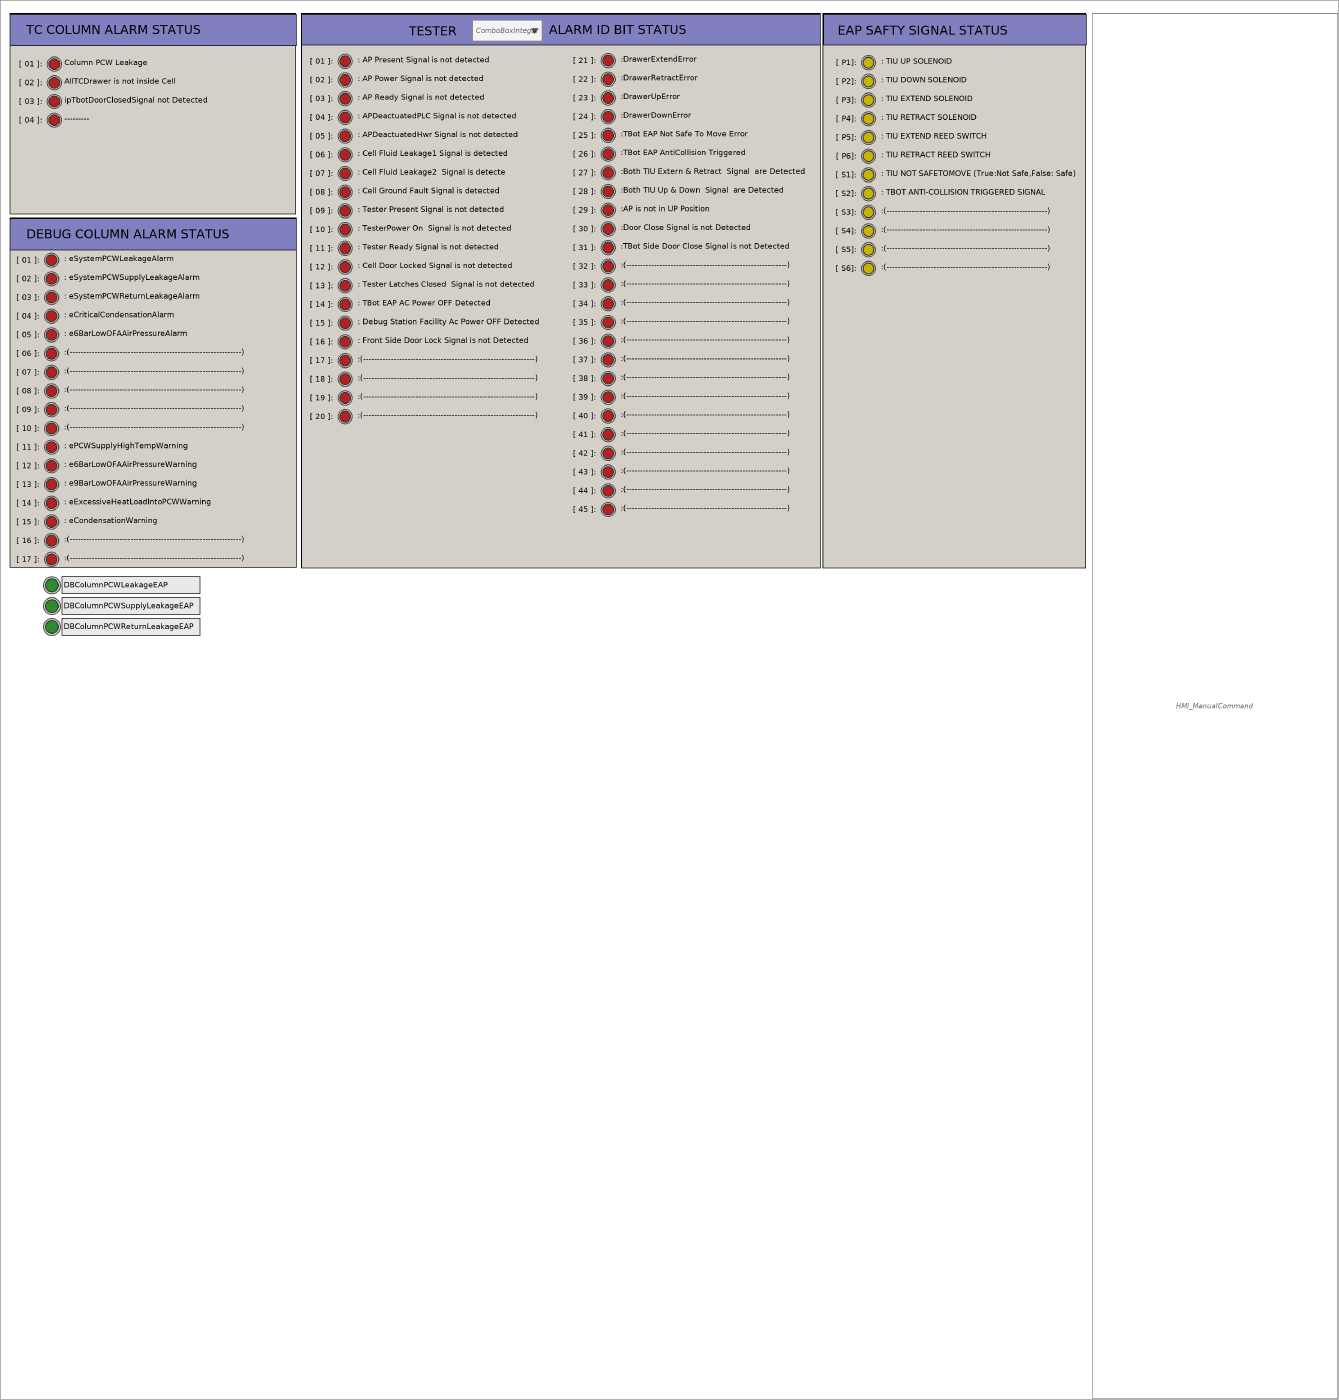
VISUALIZATION HMI_Alarm  // 1934x2021
    Rectangle (1188,19 380x801)
    Rectangle (1189,20 380x45)
    Rectangle (435,19 750x801)
    Rectangle (435,20 750x45)
    Rectangle (14,19 413x290)
    Rectangle (14,20 414x46)
    Lamp1 (866,75 25x25), variable: ALMTC.Level[iHMICbLevelSelection].AlarmID[21], style: Lamp-Lamp1-Red
    Label (824,75 40x25), "[ 21 ]:"
    Label (890,73 300x25), ":DrawerExtendError"
    ComboBoxInteger (682,29 101x30), variable: iHMICbLevelSelection, text list: 'LevelTxtList'
    Lamp1 (866,102 25x25), variable: ALMTC.Level[iHMICbLevelSelection].AlarmID[22], style: Lamp-Lamp1-Red
    Label (824,102 40x25), "[ 22 ]:"
    Label (890,100 300x25), ":DrawerRetractError"
    Lamp1 (866,129 25x25), variable: ALMTC.Level[iHMICbLevelSelection].AlarmID[23], style: Lamp-Lamp1-Red
    Label (824,129 40x25), "[ 23 ]:"
    Label (890,127 300x25), ":DrawerUpError"
    Lamp1 (866,156 25x25), variable: ALMTC.Level[iHMICbLevelSelection].AlarmID[24], style: Lamp-Lamp1-Red
    Label (824,156 40x25), "[ 24 ]:"
    Label (890,154 300x25), ":DrawerDownError"
    Lamp1 (866,183 25x25), variable: ALMTC.Level[iHMICbLevelSelection].AlarmID[25], style: Lamp-Lamp1-Red
    Label (824,183 40x25), "[ 25 ]:"
    Label (890,181 300x25), ":TBot EAP Not Safe To Move Error"
    Lamp1 (866,210 25x25), variable: ALMTC.Level[iHMICbLevelSelection].AlarmID[26], style: Lamp-Lamp1-Red
    Label (824,210 40x25), "[ 26 ]:"
    Label (890,208 300x25), ":TBot EAP AntiCollision Triggered"
    Lamp1 (866,237 25x25), variable: ALMTC.Level[iHMICbLevelSelection].AlarmID[27], style: Lamp-Lamp1-Red
    Label (824,237 40x25), "[ 27 ]:"
    Label (890,235 300x25), ":Both TIU Extern & Retract Signal are Detected"
    Lamp1 (866,264 25x25), variable: ALMTC.Level[iHMICbLevelSelection].AlarmID[28], style: Lamp-Lamp1-Red
    Label (824,264 40x25), "[ 28 ]:"
    Label (890,262 300x25), ":Both TIU Up & Down Signal are Detected"
    Lamp1 (866,291 25x25), variable: ALMTC.Level[iHMICbLevelSelection].AlarmID[29], style: Lamp-Lamp1-Red
    Label (824,291 40x25), "[ 29 ]:"
    Label (890,289 300x25), ":AP is not in UP Position"
    Lamp1 (866,318 25x25), variable: ALMTC.Level[iHMICbLevelSelection].AlarmID[30], style: Lamp-Lamp1-Red
    Label (824,318 40x25), "[ 30 ]:"
    Label (890,316 300x25), ":Door Close Signal is not Detected"
    Lamp1 (866,345 25x25), variable: ALMTC.Level[iHMICbLevelSelection].AlarmID[31], style: Lamp-Lamp1-Red
    Label (824,345 40x25), "[ 31 ]:"
    Label (890,343 300x25), ":TBot Side Door Close Signal is not Detected"
    Lamp1 (866,372 25x25), variable: ALMTC.Level[iHMICbLevelSelection].AlarmID[32], style: Lamp-Lamp1-Red
    Label (824,372 40x25), "[ 32 ]:"
    Label (890,370 300x25), ":(----------------------------------------------------------)"
    Lamp1 (866,399 25x25), variable: ALMTC.Level[iHMICbLevelSelection].AlarmID[33], style: Lamp-Lamp1-Red
    Label (824,399 40x25), "[ 33 ]:"
    Label (890,397 300x25), ":(----------------------------------------------------------)"
    Lamp1 (866,426 25x25), variable: ALMTC.Level[iHMICbLevelSelection].AlarmID[34], style: Lamp-Lamp1-Red
    Label (824,426 40x25), "[ 34 ]:"
    Label (890,424 300x25), ":(----------------------------------------------------------)"
    Lamp1 (866,453 25x25), variable: ALMTC.Level[iHMICbLevelSelection].AlarmID[35], style: Lamp-Lamp1-Red
    Label (824,453 40x25), "[ 35 ]:"
    Label (890,451 300x25), ":(----------------------------------------------------------)"
    Lamp1 (866,480 25x25), variable: ALMTC.Level[iHMICbLevelSelection].AlarmID[36], style: Lamp-Lamp1-Red
    Label (824,480 40x25), "[ 36 ]:"
    Label (890,478 300x25), ":(----------------------------------------------------------)"
    Lamp1 (866,507 25x25), variable: ALMTC.Level[iHMICbLevelSelection].AlarmID[37], style: Lamp-Lamp1-Red
    Label (824,507 40x25), "[ 37 ]:"
    Label (890,505 300x25), ":(----------------------------------------------------------)"
    Lamp1 (866,534 25x25), variable: ALMTC.Level[iHMICbLevelSelection].AlarmID[38], style: Lamp-Lamp1-Red
    Label (824,534 40x25), "[ 38 ]:"
    Label (890,532 300x25), ":(----------------------------------------------------------)"
    Lamp1 (866,561 25x25), variable: ALMTC.Level[iHMICbLevelSelection].AlarmID[39], style: Lamp-Lamp1-Red
    Label (824,561 40x25), "[ 39 ]:"
    Label (890,559 300x25), ":(----------------------------------------------------------)"
    Lamp1 (866,588 25x25), variable: ALMTC.Level[iHMICbLevelSelection].AlarmID[40], style: Lamp-Lamp1-Red
    Label (824,588 40x25), "[ 40 ]:"
    Label (890,586 300x25), ":(----------------------------------------------------------)"
    Lamp1 (866,615 25x25), variable: ALMTC.Level[iHMICbLevelSelection].AlarmID[41], style: Lamp-Lamp1-Red
    Label (824,615 40x25), "[ 41 ]:"
    Label (890,613 300x25), ":(----------------------------------------------------------)"
    Lamp1 (866,642 25x25), variable: ALMTC.Level[iHMICbLevelSelection].AlarmID[42], style: Lamp-Lamp1-Red
    Label (824,642 40x25), "[ 42 ]:"
    Label (890,640 300x25), ":(----------------------------------------------------------)"
    Lamp1 (866,669 25x25), variable: ALMTC.Level[iHMICbLevelSelection].AlarmID[43], style: Lamp-Lamp1-Red
    Label (824,669 40x25), "[ 43 ]:"
    Label (890,667 300x25), ":(----------------------------------------------------------)"
    Lamp1 (866,696 25x25), variable: ALMTC.Level[iHMICbLevelSelection].AlarmID[44], style: Lamp-Lamp1-Red
    Label (824,696 40x25), "[ 44 ]:"
    Label (890,694 300x25), ":(----------------------------------------------------------)"
    Lamp1 (866,723 25x25), variable: ALMTC.Level[iHMICbLevelSelection].AlarmID[45], style: Lamp-Lamp1-Red
    Label (824,723 40x25), "[ 45 ]:"
    Label (890,721 300x25), ":(----------------------------------------------------------)"
    Lamp1 (486,76 25x25), variable: ALMTC.Level[iHMICbLevelSelection].AlarmID[1], style: Lamp-Lamp1-Red
    Label (444,76 40x25), "[ 01 ]:"
    Label (510,74 300x25), ": AP Present Signal is not detected"
    Lamp1 (486,103 25x25), variable: ALMTC.Level[iHMICbLevelSelection].AlarmID[2], style: Lamp-Lamp1-Red
    Label (444,103 40x25), "[ 02 ]:"
    Label (510,101 300x25), ": AP Power Signal is not detected"
    Lamp1 (486,130 25x25), variable: ALMTC.Level[iHMICbLevelSelection].AlarmID[3], style: Lamp-Lamp1-Red
    Label (444,130 40x25), "[ 03 ]:"
    Label (510,128 300x25), ": AP Ready Signal is not detected"
    Lamp1 (486,157 25x25), variable: ALMTC.Level[iHMICbLevelSelection].AlarmID[4], style: Lamp-Lamp1-Red
    Label (444,157 40x25), "[ 04 ]:"
    Label (510,155 300x25), ": APDeactuatedPLC Signal is not detected"
    Lamp1 (486,184 25x25), variable: ALMTC.Level[iHMICbLevelSelection].AlarmID[5], style: Lamp-Lamp1-Red
    Label (444,184 40x25), "[ 05 ]:"
    Label (510,182 300x25), ": APDeactuatedHwr Signal is not detected"
    Lamp1 (486,211 25x25), variable: ALMTC.Level[iHMICbLevelSelection].AlarmID[6], style: Lamp-Lamp1-Red
    Label (444,211 40x25), "[ 06 ]:"
    Label (510,209 300x25), ": Cell Fluid Leakage1 Signal is detected"
    Lamp1 (486,238 25x25), variable: ALMTC.Level[iHMICbLevelSelection].AlarmID[7], style: Lamp-Lamp1-Red
    Label (444,238 40x25), "[ 07 ]:"
    Label (510,236 300x25), ": Cell Fluid Leakage2 Signal is detecte"
    Lamp1 (486,265 25x25), variable: ALMTC.Level[iHMICbLevelSelection].AlarmID[8], style: Lamp-Lamp1-Red
    Label (444,265 40x25), "[ 08 ]:"
    Label (510,263 300x25), ": Cell Ground Fault Signal is detected"
    Lamp1 (486,292 25x25), variable: ALMTC.Level[iHMICbLevelSelection].AlarmID[9], style: Lamp-Lamp1-Red
    Label (444,292 40x25), "[ 09 ]:"
    Label (510,290 300x25), ": Tester Present Signal is not detected"
    Lamp1 (486,319 25x25), variable: ALMTC.Level[iHMICbLevelSelection].AlarmID[10], style: Lamp-Lamp1-Red
    Label (444,319 40x25), "[ 10 ]:"
    Label (510,317 300x25), ": TesterPower On Signal is not detected"
    Lamp1 (486,346 25x25), variable: ALMTC.Level[iHMICbLevelSelection].AlarmID[11], style: Lamp-Lamp1-Red
    Label (444,346 40x25), "[ 11 ]:"
    Label (510,344 300x25), ": Tester Ready Signal is not detected"
    Lamp1 (486,373 25x25), variable: ALMTC.Level[iHMICbLevelSelection].AlarmID[12], style: Lamp-Lamp1-Red
    Label (444,373 40x25), "[ 12 ]:"
    Label (510,371 300x25), ": Cell Door Locked Signal is not detected"
    Lamp1 (486,400 25x25), variable: ALMTC.Level[iHMICbLevelSelection].AlarmID[13], style: Lamp-Lamp1-Red
    Label (444,400 40x25), "[ 13 ]:"
    Label (510,398 300x25), ": Tester Latches Closed Signal is not detected"
    Lamp1 (486,427 25x25), variable: ALMTC.Level[iHMICbLevelSelection].AlarmID[14], style: Lamp-Lamp1-Red
    Label (444,427 40x25), "[ 14 ]:"
    Label (510,425 300x25), ": TBot EAP AC Power OFF Detected"
    Lamp1 (486,454 25x25), variable: ALMTC.Level[iHMICbLevelSelection].AlarmID[15], style: Lamp-Lamp1-Red
    Label (444,454 40x25), "[ 15 ]:"
    Label (510,452 300x25), ": Debug Station Facility Ac Power OFF Detected"
    Lamp1 (486,481 25x25), variable: ALMTC.Level[iHMICbLevelSelection].AlarmID[16], style: Lamp-Lamp1-Red
    Label (444,481 40x25), "[ 16 ]:"
    Label (510,479 300x25), ": Front Side Door Lock Signal is not Detected"
    Lamp1 (486,508 25x25), variable: ALMTC.Level[iHMICbLevelSelection].AlarmID[17], style: Lamp-Lamp1-Red
    Label (444,508 40x25), "[ 17 ]:"
    Label (510,506 300x25), ":(--------------------------------------------------------------)"
    Lamp1 (486,535 25x25), variable: ALMTC.Level[iHMICbLevelSelection].AlarmID[18], style: Lamp-Lamp1-Red
    Label (444,535 40x25), "[ 18 ]:"
    Label (510,533 300x25), ":(--------------------------------------------------------------)"
    Lamp1 (486,562 25x25), variable: ALMTC.Level[iHMICbLevelSelection].AlarmID[19], style: Lamp-Lamp1-Red
    Label (444,562 40x25), "[ 19 ]:"
    Label (510,560 300x25), ":(--------------------------------------------------------------)"
    Lamp1 (486,589 25x25), variable: ALMTC.Level[iHMICbLevelSelection].AlarmID[20], style: Lamp-Lamp1-Red
    Label (444,589 40x25), "[ 20 ]:"
    Label (510,587 300x25), ":(--------------------------------------------------------------)"
    Lamp1 (66,80 25x25), variable: ALMTC.Common.AlarmID[1], style: Lamp-Lamp1-Red
    Label (24,80 40x25), "[ 01 ]:"
    Label (90,78 300x25), "Column PCW Leakage"
    Lamp1 (66,107 25x25), variable: ALMTC.Common.AlarmID[2], style: Lamp-Lamp1-Red
    Label (24,107 40x25), "[ 02 ]:"
    Label (90,105 300x25), "AllTCDrawer is not inside Cell"
    Lamp1 (66,134 25x25), variable: ALMTC.Common.AlarmID[3], style: Lamp-Lamp1-Red
    Label (24,134 40x25), "[ 03 ]:"
    Label (90,132 300x25), "ipTbotDoorClosedSignal not Detected"
    Lamp1 (66,161 25x25), variable: ALMTC.Common.AlarmID[4], style: Lamp-Lamp1-Red
    Label (24,161 40x25), "[ 04 ]:"
    Label (90,159 300x25), "---------"
    Label (587,25 81x40), "TESTER"
    Label (790,23 243x40), "ALARM ID BIT STATUS"
    Label (35,23 388x40), "TC COLUMN ALARM STATUS"
    Lamp1 (1242,78 25x25), style: Lamp-Lamp1-Yellow
    Label (1200,78 40x25), "[ P1]:"
    Label (1266,76 300x25), ": TIU UP SOLENOID"
    Lamp1 (1242,105 25x25), style: Lamp-Lamp1-Yellow
    Label (1200,105 40x25), "[ P2]:"
    Label (1266,103 300x25), ": TIU DOWN SOLENOID"
    Lamp1 (1242,132 25x25), style: Lamp-Lamp1-Yellow
    Label (1200,132 40x25), "[ P3]:"
    Label (1266,130 300x25), ": TIU EXTEND SOLENOID"
    Lamp1 (1242,159 25x25), style: Lamp-Lamp1-Yellow
    Label (1200,159 40x25), "[ P4]:"
    Label (1266,157 300x25), ": TIU RETRACT SOLENOID"
    Lamp1 (1242,186 25x25), style: Lamp-Lamp1-Yellow
    Label (1200,186 40x25), "[ P5]:"
    Label (1266,184 300x25), ": TIU EXTEND REED SWITCH"
    Lamp1 (1242,213 25x25), style: Lamp-Lamp1-Yellow
    Label (1200,213 40x25), "[ P6]:"
    Label (1266,211 300x25), ": TIU RETRACT REED SWITCH"
    Lamp1 (1242,240 25x25), variable: stEAP.stTBOT_TC_EAP[iHMICbLevelSelection].iTCDwrSafeToMoveEAP, style: Lamp-Lamp1-Yellow
    Label (1200,240 40x25), "[ S1]:"
    Label (1266,238 300x25), ": TIU NOT SAFETOMOVE (True:Not Safe,False: Safe)"
    Lamp1 (1242,267 25x25), variable: stEAP.stTBOT_TC_EAP[iHMICbLevelSelection].bAntiCollisionTriggered, style: Lamp-Lamp1-Yellow
    Label (1200,267 40x25), "[ S2]:"
    Label (1266,265 300x25), ": TBOT ANTI-COLLISION TRIGGERED SIGNAL"
    Lamp1 (1242,294 25x25), style: Lamp-Lamp1-Yellow
    Label (1200,294 40x25), "[ S3]:"
    Label (1266,292 300x25), ":(----------------------------------------------------------)"
    Lamp1 (1242,321 25x25), style: Lamp-Lamp1-Yellow
    Label (1200,321 40x25), "[ S4]:"
    Label (1266,319 300x25), ":(----------------------------------------------------------)"
    Lamp1 (1242,348 25x25), style: Lamp-Lamp1-Yellow
    Label (1200,348 40x25), "[ S5]:"
    Label (1266,346 300x25), ":(----------------------------------------------------------)"
    Lamp1 (1242,375 25x25), style: Lamp-Lamp1-Yellow
    Label (1200,375 40x25), "[ S6]:"
    Label (1266,373 300x25), ":(----------------------------------------------------------)"
    Label (1207,24 305x40), "EAP SAFTY SIGNAL STATUS"
    Rectangle (14,314 414x505)
    Rectangle (14,315 414x46)
    Label (35,318 388x40), "DEBUG COLUMN ALARM STATUS"
    Lamp1 (62,363 25x25), variable: ALM_DCCOL.AlarmID[1], style: Lamp-Lamp1-Red
    Label (20,363 40x25), "[ 01 ]:"
    Label (86,361 300x25), ": eSystemPCWLeakageAlarm"
    Lamp1 (62,390 25x25), variable: ALM_DCCOL.AlarmID[2], style: Lamp-Lamp1-Red
    Label (20,390 40x25), "[ 02 ]:"
    Label (86,388 300x25), ": eSystemPCWSupplyLeakageAlarm"
    Lamp1 (62,417 25x25), variable: ALM_DCCOL.AlarmID[3], style: Lamp-Lamp1-Red
    Label (20,417 40x25), "[ 03 ]:"
    Label (86,415 300x25), ": eSystemPCWReturnLeakageAlarm"
    Lamp1 (62,444 25x25), variable: ALM_DCCOL.AlarmID[4], style: Lamp-Lamp1-Red
    Label (20,444 40x25), "[ 04 ]:"
    Label (86,442 300x25), ": eCriticalCondensationAlarm"
    Lamp1 (62,471 25x25), variable: ALM_DCCOL.AlarmID[5], style: Lamp-Lamp1-Red
    Label (20,471 40x25), "[ 05 ]:"
    Label (86,469 300x25), ": e6BarLowOFAAirPressureAlarm"
    Lamp1 (62,498 25x25), variable: ALM_DCCOL.AlarmID[6], style: Lamp-Lamp1-Red
    Label (20,498 40x25), "[ 06 ]:"
    Label (86,496 300x25), ":(--------------------------------------------------------------)"
    Lamp1 (62,525 25x25), variable: ALM_DCCOL.AlarmID[7], style: Lamp-Lamp1-Red
    Label (20,525 40x25), "[ 07 ]:"
    Label (86,523 300x25), ":(--------------------------------------------------------------)"
    Lamp1 (62,552 25x25), variable: ALM_DCCOL.AlarmID[8], style: Lamp-Lamp1-Red
    Label (20,552 40x25), "[ 08 ]:"
    Label (86,550 300x25), ":(--------------------------------------------------------------)"
    Lamp1 (62,579 25x25), variable: ALM_DCCOL.AlarmID[9], style: Lamp-Lamp1-Red
    Label (20,579 40x25), "[ 09 ]:"
    Label (86,577 300x25), ":(--------------------------------------------------------------)"
    Lamp1 (62,606 25x25), variable: ALM_DCCOL.AlarmID[10], style: Lamp-Lamp1-Red
    Label (20,606 40x25), "[ 10 ]:"
    Label (86,604 300x25), ":(--------------------------------------------------------------)"
    Lamp1 (62,633 25x25), variable: ALM_DCCOL.AlarmID[11], style: Lamp-Lamp1-Red
    Label (20,633 40x25), "[ 11 ]:"
    Label (86,631 300x25), ": ePCWSupplyHighTempWarning"
    Lamp1 (62,660 25x25), variable: ALM_DCCOL.AlarmID[12], style: Lamp-Lamp1-Red
    Label (20,660 40x25), "[ 12 ]:"
    Label (86,658 300x25), ": e6BarLowOFAAirPressureWarning"
    Lamp1 (62,687 25x25), variable: ALM_DCCOL.AlarmID[13], style: Lamp-Lamp1-Red
    Label (20,687 40x25), "[ 13 ]:"
    Label (86,685 300x25), ": e9BarLowOFAAirPressureWarning"
    Lamp1 (62,714 25x25), variable: ALM_DCCOL.AlarmID[14], style: Lamp-Lamp1-Red
    Label (20,714 40x25), "[ 14 ]:"
    Label (86,712 300x25), ": eExcessiveHeatLoadIntoPCWWarning"
    Lamp1 (62,741 25x25), variable: ALM_DCCOL.AlarmID[15], style: Lamp-Lamp1-Red
    Label (20,741 40x25), "[ 15 ]:"
    Label (86,739 300x25), ": eCondensationWarning"
    Lamp1 (62,768 25x25), variable: ALM_DCCOL.AlarmID[16], style: Lamp-Lamp1-Red
    Label (20,768 40x25), "[ 16 ]:"
    Label (86,766 300x25), ":(--------------------------------------------------------------)"
    Lamp1 (62,795 25x25), variable: ALM_DCCOL.AlarmID[17], style: Lamp-Lamp1-Red
    Label (20,795 40x25), "[ 17 ]:"
    Label (86,793 300x25), ":(--------------------------------------------------------------)"
    RoundedRectangle (89,832 200x25), "DBColumnPCWLeakageEAP"
        toggle fbDebugColumn.stDebugColumnDIO.eapDBColumnPCWLeakage
    Lamp1 (60,830 30x30), variable: fbDebugColumn.stDebugColumnDIO.eapDBColumnPCWLeakage, style: Lamp-Lamp1-Green
    RoundedRectangle (89,862 200x25), "DBColumnPCWSupplyLeakageEAP"
        toggle fbDebugColumn.stDebugColumnDIO.eapDBColumnPCWSupplyLeakage
    Lamp1 (60,860 30x30), variable: fbDebugColumn.stDebugColumnDIO.eapDBColumnPCWSupplyLeakage, style: Lamp-Lamp1-Green
    RoundedRectangle (89,892 200x25), "DBColumnPCWReturnLeakageEAP"
        toggle fbDebugColumn.stDebugColumnDIO.eapDBColumnPCWReturnLeakage
    Lamp1 (60,890 30x30), variable: fbDebugColumn.stDebugColumnDIO.eapDBColumnPCWReturnLeakage, style: Lamp-Lamp1-Green
    Frame (1577,19 355x2000), invisible if: Not bEnableManualCommandTest1 AND Not bEnableManualCommandTest2
        shows HMI_ManualCommand()
END_VISUALIZATION

(* stored: Version 1.1.0.1, ProductVersion 3.1.4022.18
   Visu HMI_Alarm: Id {f9e8604f-fcf7-4035-8450-110c1ad232b7} *)
